(* CoDeSys 2.3.9.59 project: Nastro_Timer, Contatore e Pulsante.pro *)
(* Libraries: STANDARD.LIB *)

(* Task configuration *)
TASK Standard (PRIORITY := 0, INTERVAL := T#10ms);
	MAIN
END_TASK

(* POU MAIN, LD *)
PROGRAM MAIN
VAR

	pezzo_magazzino  AT%IX0.0:BOOL;
	fine_corsa_nastro  AT%IX0.6:BOOL;
	pistone_avanti AT%IX0.2:BOOL;
	pistone_indietro AT%IX0.4:BOOL;
	pulsante:BOOL;
         reset:BOOL;

	nastro_on  AT%QX0.0:BOOL;
	pistone_on  AT%QX0.2:BOOL;
	timer:BOOL;

	timer_nastro: TON;
	mytime: TIME;

	conta_pezzi_nastro: CTU;
	mycounter: REAL;
	contatore: BOOL;

END_VAR
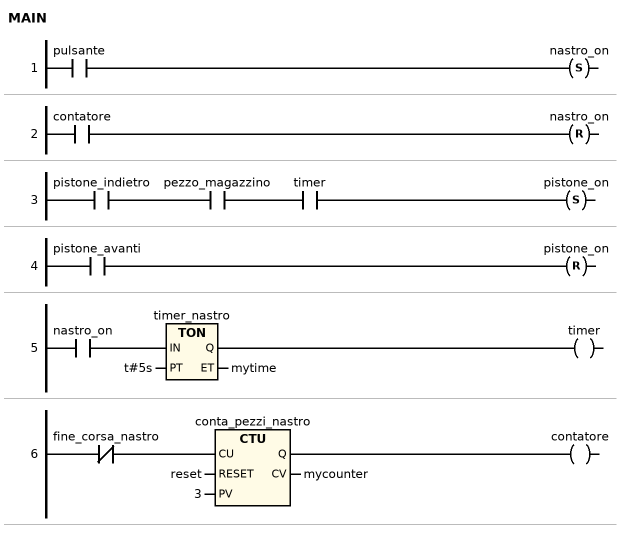
_LD_ (* Ladder Diagram *)
NETWORK 1
	[pulsante] --- (S nastro_on)
NETWORK 2
	[contatore] --- (R nastro_on)
NETWORK 3
	[pistone_indietro] - [pezzo_magazzino] - [timer] --- (S pistone_on)
NETWORK 4
	[pistone_avanti] --- (R pistone_on)
NETWORK 5
	[nastro_on] - timer_nastro:TON(IN: *, PT: t#5s, ET => mytime) --- (timer)
NETWORK 6
	[/fine_corsa_nastro] - conta_pezzi_nastro:CTU(CU: *, RESET: reset, PV: 3, CV => mycounter) --- (contatore)
_END_LD_
(* the same logic as Structured Text *)
(* Network 1 *)
IF pulsante THEN nastro_on := TRUE; END_IF;
(* Network 2 *)
IF contatore THEN nastro_on := FALSE; END_IF;
(* Network 3 *)
IF pistone_indietro AND pezzo_magazzino AND timer THEN pistone_on := TRUE; END_IF;
(* Network 4 *)
IF pistone_avanti THEN pistone_on := FALSE; END_IF;
(* Network 5 *)
timer_nastro(IN := nastro_on, PT := t#5s);
mytime := timer_nastro.ET;
timer := timer_nastro.Q;
(* Network 6 *)
conta_pezzi_nastro(CU := NOT fine_corsa_nastro, RESET := reset, PV := 3);
mycounter := conta_pezzi_nastro.CV;
contatore := conta_pezzi_nastro.Q;
END_PROGRAM

(* Visualisation prova
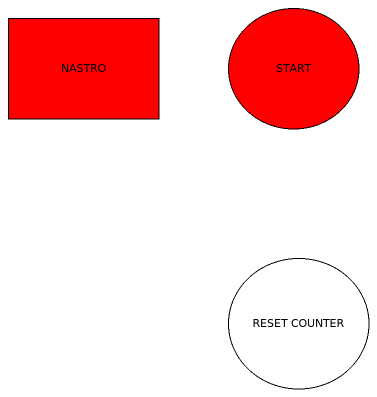
ellipse at (270,60)-(401,181): text "START"; toggles MAIN.nastro_on
rounded rectangle at (50,70)-(201,171): text "NASTRO"; alarm colour if MAIN.nastro_on
ellipse at (270,310)-(411,441): text "RESET COUNTER"; taps MAIN.reset
*)
